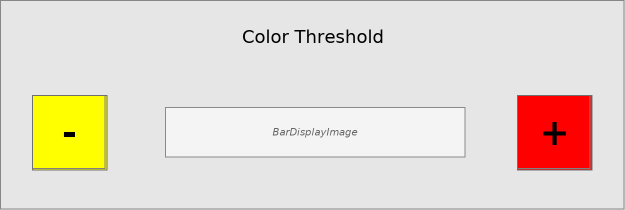
VISUALIZATION ColorThreshold  // 625x210
    Button (517,95 75x75), "+"
    Button (32,95 75x75), "-"
    Textfield (238,22 150x30), "Color Threshold"
    BarDisplayImage (165,107 300x50), style: BarDisplayImage-Gray, scale format: %.1f, scale 0..100
END_VISUALIZATION

(* stored: Version 1.1.0.1, ProductVersion 3.1.4024.15
   Visu ColorThreshold: Id {dc07d54b-1c50-4435-a6b4-a182c5472fc8} *)
